# EPICS autosave request: iocBoot/iocUSB3105/auto_settings.req
file "USB2408_settings.req", P=$(P)
